TYPE ST_CsvTableRowData :
STRUCT
	sTimeStamp:STRING;
	sDescription:STRING;
	sValue:STRING;
	sUnit:STRING;
END_STRUCT
END_TYPE

(* stored: Version 1.1.0.1, ProductVersion 3.1.4024.12
   DUT ST_CsvTableRowData: Id {1f3413b8-ca74-4ea8-8e15-7af148e6f828} *)
